# EPICS autosave request: ipApp/Db/PTC10_coldj_chan_settings.req
$(P)$(T):$(C):temperature.SCAN
